(* PLC project mtcs_telemetry, Institute of Astronomy Onto 0.0.1 *)
(* stored: creationDateTime 2024-10-01T22:53:32.010142, modificationDateTime 2024-10-01T22:53:32.010142 *)

TYPE TelemetryParts : STRUCT
  temperatures : TelemetryTemperatures;  (* All temperature measurements *)
  relativeHumidities : TelemetryRelativeHumidities;  (* All relative humidity measurements *)
  dewpoints : TelemetryDewpoints;  (* All calculated dewpoints *)
  accelerometers : TelemetryAccelerometers;  (* Feedback from the accelerometers (vibrations + angles) *)
  io : TelemetryIO;  (* I/O modules *)
  flatfieldLeds : TelemetryFlatfieldLeds;  (* I/O modules *)
  configManager : ConfigManager;  (* The config manager (to load/save/activate configuration data) *)
END_STRUCT;
END_TYPE

TYPE TelemetryFlatfieldLedsParts : STRUCT
  output1 : SimpleRelay;  (* Output 1 *)
  output2 : SimpleRelay;  (* Output 2 *)
  output3 : SimpleRelay;  (* Output 3 *)
  output4 : SimpleRelay;  (* Output 4 *)
  output5 : SimpleRelay;  (* Output 5 *)
  output6 : SimpleRelay;  (* Output 6 *)
  output7 : SimpleRelay;  (* Output 7 *)
  output8 : SimpleRelay;  (* Output 8 *)
END_STRUCT;
END_TYPE

TYPE TelemetryIOParts : STRUCT
  coupler : EtherCatDevice;  (* Coupler *)
  slot5 : EtherCatDevice;  (* Slot 5 *)
  slot6 : EtherCatDevice;  (* Slot 6 *)
  slot7 : EtherCatDevice;  (* Slot 7 *)
  slot8 : EtherCatDevice;  (* Slot 8 *)
  slot9 : EtherCatDevice;  (* Slot 9 *)
  slot10 : EtherCatDevice;  (* Slot 10 *)
  slot11 : EtherCatDevice;  (* Slot 11 *)
  slot12 : EtherCatDevice;  (* Slot 12 *)
  slot13 : EtherCatDevice;  (* Slot 13 *)
  tubeAccelerometers : EtherCatDevice;  (* Tube accelerometers *)
END_STRUCT;
END_TYPE

TYPE TelemetryProcesses : STRUCT
  initialize : Process;  (* Start initializing *)
  lock : Process;  (* Lock the system *)
  unlock : Process;  (* Unlock the system *)
  changeOperatingState : ChangeOperatingStateProcess;  (* Change the operating state (e.g. AUTO, MANUAL, ...) *)
END_STRUCT;
END_TYPE

TYPE TelemetryTemperaturesStatuses : STRUCT
  healthStatus : HealthStatus;  (* Are all temperatures in a healthy state? *)
END_STRUCT;
END_TYPE

TYPE TelemetryRelativeHumiditiesStatuses : STRUCT
  healthStatus : HealthStatus;  (* Are all relative humidities in a healthy state? *)
END_STRUCT;
END_TYPE

TYPE TelemetryDewpointStatuses : STRUCT
  enabledStatus : EnabledStatus;  (* Is the dewpoint being calculated? *)
  healthStatus : HealthStatus;  (* Is the depoint OK? *)
  alarmStatus : HiHiLoLoAlarmStatus;  (* Alarm status *)
END_STRUCT;
END_TYPE

TYPE TelemetryDewpointsStatuses : STRUCT
  healthStatus : HealthStatus;  (* Are all dewpoints in a healthy state? *)
END_STRUCT;
END_TYPE

TYPE TelemetryAccelerometerStatuses : STRUCT
  xEnabledStatus : EnabledStatus;  (* Is the X angle being measured? *)
  yEnabledStatus : EnabledStatus;  (* Is the Y angle being measured? *)
  xHealthStatus : HealthStatus;  (* Is the X angle measurement OK? *)
  yHealthStatus : HealthStatus;  (* Is the Y angle measurement OK? *)
  xAlarmStatus : HiHiLoLoAlarmStatus;  (* Alarm status of the X angle *)
  yAlarmStatus : HiHiLoLoAlarmStatus;  (* Alarm status of the Y angle *)
END_STRUCT;
END_TYPE

TYPE TelemetryAccelerometersStatuses : STRUCT
  healthStatus : HealthStatus;  (* Are all accelerometers in a healthy state? *)
END_STRUCT;
END_TYPE

TYPE TelemetryStatuses : STRUCT
  initializationStatus : InitializationStatus;
  healthStatus : HealthStatus;
  busyStatus : BusyStatus;
  operatingStatus : OperatingStatus;
END_STRUCT;
END_TYPE

TYPE TelemetryFlatfieldLedsStatuses : STRUCT
  busyStatus : BusyStatus;
END_STRUCT;
END_TYPE

TYPE TelemetryIOStatuses : STRUCT
  healthStatus : HealthStatus;  (* Is the I/O in a healthy state? *)
END_STRUCT;
END_TYPE

TYPE TelemetryTemperaturesConfig : STRUCT
  m1 : MeasurementConfig;  (* Temperature of M1 *)
  mirrorCell : MeasurementConfig;  (* Temperature of the mirror cell *)
  m2 : MeasurementConfig;  (* Temperature of M2 *)
  m2Electronics : MeasurementConfig;  (* Temperature of the M2 electricity *)
  topTube : MeasurementConfig;  (* Temperature of the top of the tube *)
  centreTube : MeasurementConfig;  (* Temperature of the centre of the tube *)
  fork : MeasurementConfig;  (* Temperature of the fork *)
  nasmythAir : MeasurementConfig;  (* Temperature of the air inside the Nasmyth focal station *)
  rem : MeasurementConfig;  (* Temperature inside the REM cabinet *)
  rpm : MeasurementConfig;  (* Temperature inside the RPM cabinet *)
  hermesTelescopeAdapter : MeasurementConfig;  (* Temperature inside the HERMES telescope adapter *)
  topAir : MeasurementConfig;  (* Temperature of the air at the top of the tube *)
  insideTube : MeasurementConfig;  (* Temperature of the air inside the tube *)
END_STRUCT;
END_TYPE

TYPE TelemetryRelativeHumiditiesConfig : STRUCT
  topAir : MeasurementConfig;  (* Relative humidity of the air at the top of the tube *)
  insideTube : MeasurementConfig;  (* Relative humidity of the air inside the tube *)
END_STRUCT;
END_TYPE

TYPE TelemetryDewpointsConfig : STRUCT
  topAir : MeasurementConfig;  (* Dewpoint of the air at the top of the tube *)
  insideTube : MeasurementConfig;  (* Dewpoint of the air inside the tube *)
END_STRUCT;
END_TYPE

TYPE TelemetryAccelerometerConfig : STRUCT
  x : MeasurementConfig;  (* X angle *)
  y : MeasurementConfig;  (* X angle *)
END_STRUCT;
END_TYPE

TYPE TelemetryAccelerometersConfig : STRUCT
  tube : TelemetryAccelerometerConfig;  (* Accelerometer box at the tube *)
END_STRUCT;
END_TYPE

TYPE TelemetryConfig : STRUCT
  temperatures : TelemetryTemperaturesConfig;  (* All temperatures *)
  relativeHumidities : TelemetryRelativeHumiditiesConfig;  (* All relative humidities *)
  dewpoints : TelemetryDewpointsConfig;  (* All dewpoints *)
  accelerometers : TelemetryAccelerometersConfig;  (* All accelerometers *)
END_STRUCT;
END_TYPE

FUNCTION_BLOCK SM_TelemetryTemperatures
  VAR_OUTPUT
    {attribute 'OPC.UA.DA' := '1'}
    {attribute 'OPC.UA.DA.Access' := '1'}
    actualStatus : STRING;  (* Current status description *)
    previousStatus : STRING;  (* Previous status description *)
    {attribute 'OPC.UA.DA' := '1'}
    {attribute 'OPC.UA.DA.Access' := '1'}
    m1 : TemperatureMeasurement;  (* Temperature of M1 *)
    {attribute 'OPC.UA.DA' := '1'}
    {attribute 'OPC.UA.DA.Access' := '1'}
    mirrorCell : TemperatureMeasurement;  (* Temperature of the mirror cell *)
    {attribute 'OPC.UA.DA' := '1'}
    {attribute 'OPC.UA.DA.Access' := '1'}
    m2 : TemperatureMeasurement;  (* Temperature of M2 *)
    {attribute 'OPC.UA.DA' := '1'}
    {attribute 'OPC.UA.DA.Access' := '1'}
    m2Electronics : TemperatureMeasurement;  (* Temperature of the M2 electricity *)
    {attribute 'OPC.UA.DA' := '1'}
    {attribute 'OPC.UA.DA.Access' := '1'}
    topTube : TemperatureMeasurement;  (* Temperature of the top of the tube *)
    {attribute 'OPC.UA.DA' := '1'}
    {attribute 'OPC.UA.DA.Access' := '1'}
    centreTube : TemperatureMeasurement;  (* Temperature of the centre of the tube *)
    {attribute 'OPC.UA.DA' := '1'}
    {attribute 'OPC.UA.DA.Access' := '1'}
    fork : TemperatureMeasurement;  (* Temperature of the fork *)
    {attribute 'OPC.UA.DA' := '1'}
    {attribute 'OPC.UA.DA.Access' := '1'}
    nasmythAir : TemperatureMeasurement;  (* Temperature of the air inside the Nasmyth focal station *)
    {attribute 'OPC.UA.DA' := '1'}
    {attribute 'OPC.UA.DA.Access' := '1'}
    rem : TemperatureMeasurement;  (* Temperature inside the REM cabinet *)
    {attribute 'OPC.UA.DA' := '1'}
    {attribute 'OPC.UA.DA.Access' := '1'}
    rpm : TemperatureMeasurement;  (* Temperature inside the RPM cabinet *)
    {attribute 'OPC.UA.DA' := '1'}
    {attribute 'OPC.UA.DA.Access' := '1'}
    hermesTelescopeAdapter : TemperatureMeasurement;  (* Temperature inside the HERMES telescope adapter *)
    {attribute 'OPC.UA.DA' := '1'}
    {attribute 'OPC.UA.DA.Access' := '1'}
    topAir : TemperatureMeasurement;  (* Temperature of the air at the top of the tube *)
    {attribute 'OPC.UA.DA' := '1'}
    {attribute 'OPC.UA.DA.Access' := '1'}
    insideTube : TemperatureMeasurement;  (* Temperature of the air inside the tube *)
    statuses : TelemetryTemperaturesStatuses;  (* Statuses of the state machine *)
  END_VAR
  VAR_IN_OUT
    {attribute 'OPC.UA.DA' := '0'}
    config : TelemetryTemperaturesConfig;  (* Configuration of the temperatures *)
  END_VAR

            m1( config := config.m1 );
mirrorCell( config := config.mirrorCell );
m2( config := config.m2 );
m2Electronics( config := config.m2Electronics );
topTube( config := config.topTube );
centreTube( config := config.centreTube );
fork( config := config.fork );
nasmythAir( config := config.nasmythAir );
rem( config := config.rem );
rpm( config := config.rpm );
hermesTelescopeAdapter( config := config.hermesTelescopeAdapter );
topAir( config := config.topAir );
insideTube( config := config.insideTube );
statuses.healthStatus(
    isGood := (m1.statuses.healthStatus.isGood OR m1.statuses.enabledStatus.disabled) AND ((mirrorCell.statuses.healthStatus.isGood OR mirrorCell.statuses.enabledStatus.disabled) AND ((m2.statuses.healthStatus.isGood OR m2.statuses.enabledStatus.disabled) AND ((m2Electronics.statuses.healthStatus.isGood OR m2Electronics.statuses.enabledStatus.disabled) AND ((topTube.statuses.healthStatus.isGood OR topTube.statuses.enabledStatus.disabled) AND ((centreTube.statuses.healthStatus.isGood OR centreTube.statuses.enabledStatus.disabled) AND ((fork.statuses.healthStatus.isGood OR fork.statuses.enabledStatus.disabled) AND ((nasmythAir.statuses.healthStatus.isGood OR nasmythAir.statuses.enabledStatus.disabled) AND ((rem.statuses.healthStatus.isGood OR rem.statuses.enabledStatus.disabled) AND ((rpm.statuses.healthStatus.isGood OR rpm.statuses.enabledStatus.disabled) AND ((hermesTelescopeAdapter.statuses.healthStatus.isGood OR hermesTelescopeAdapter.statuses.enabledStatus.disabled) AND ((topAir.statuses.healthStatus.isGood OR topAir.statuses.enabledStatus.disabled) AND (insideTube.statuses.healthStatus.isGood OR insideTube.statuses.enabledStatus.disabled)))))))))))),
    hasWarning := m1.statuses.healthStatus.hasWarning OR (mirrorCell.statuses.healthStatus.hasWarning OR (m2.statuses.healthStatus.hasWarning OR (m2Electronics.statuses.healthStatus.hasWarning OR (topTube.statuses.healthStatus.hasWarning OR (centreTube.statuses.healthStatus.hasWarning OR (fork.statuses.healthStatus.hasWarning OR (nasmythAir.statuses.healthStatus.hasWarning OR (rem.statuses.healthStatus.hasWarning OR (rpm.statuses.healthStatus.hasWarning OR (hermesTelescopeAdapter.statuses.healthStatus.hasWarning OR (topAir.statuses.healthStatus.hasWarning OR insideTube.statuses.healthStatus.hasWarning))))))))))));

          

{attribute 'TcRpcEnable' := '1'}
METHOD _log : BOOL
  VAR_INPUT
    name : STRING;  (* Name of this function block instance *)
  END_VAR
  VAR_IN_OUT
    buffer : LogBuffer;  (* Buffer to write all logging to *)
  END_VAR
  VAR
    subBuffer : LogBuffer;  (* Temporary buffer to write logging by parts (sub-statemachines) to *)
  END_VAR
                  LOGGER(
    name := name,
    actualStatus := THIS^.actualStatus,
    previousStatus := THIS^.previousStatus,
    buffer := buffer,
    subBuffer := subBuffer,
    pHealthStatus := ADR(THIS^.statuses.healthStatus));

                
END_METHOD
END_FUNCTION_BLOCK

FUNCTION_BLOCK SM_TelemetryRelativeHumidities
  VAR_OUTPUT
    {attribute 'OPC.UA.DA' := '1'}
    {attribute 'OPC.UA.DA.Access' := '1'}
    actualStatus : STRING;  (* Current status description *)
    previousStatus : STRING;  (* Previous status description *)
    {attribute 'OPC.UA.DA' := '1'}
    {attribute 'OPC.UA.DA.Access' := '1'}
    topAir : RelativeHumidityMeasurement;  (* Relative humidity of the air at the top of the tube *)
    {attribute 'OPC.UA.DA' := '1'}
    {attribute 'OPC.UA.DA.Access' := '1'}
    insideTube : RelativeHumidityMeasurement;  (* Relative humidity of the air inside the tube *)
    statuses : TelemetryRelativeHumiditiesStatuses;  (* Statuses of the state machine *)
  END_VAR
  VAR_IN_OUT
    {attribute 'OPC.UA.DA' := '0'}
    config : TelemetryRelativeHumiditiesConfig;  (* Configuration of the relative humidities *)
  END_VAR

            topAir( config := config.topAir );
insideTube( config := config.insideTube );
statuses.healthStatus(
    isGood := (topAir.statuses.healthStatus.isGood OR topAir.statuses.enabledStatus.disabled) AND (insideTube.statuses.healthStatus.isGood OR insideTube.statuses.enabledStatus.disabled),
    hasWarning := topAir.statuses.healthStatus.hasWarning OR insideTube.statuses.healthStatus.hasWarning);

          

{attribute 'TcRpcEnable' := '1'}
METHOD _log : BOOL
  VAR_INPUT
    name : STRING;  (* Name of this function block instance *)
  END_VAR
  VAR_IN_OUT
    buffer : LogBuffer;  (* Buffer to write all logging to *)
  END_VAR
  VAR
    subBuffer : LogBuffer;  (* Temporary buffer to write logging by parts (sub-statemachines) to *)
  END_VAR
                  LOGGER(
    name := name,
    actualStatus := THIS^.actualStatus,
    previousStatus := THIS^.previousStatus,
    buffer := buffer,
    subBuffer := subBuffer,
    pHealthStatus := ADR(THIS^.statuses.healthStatus));

                
END_METHOD
END_FUNCTION_BLOCK

FUNCTION_BLOCK SM_TelemetryDewpoint
  VAR_OUTPUT
    {attribute 'OPC.UA.DA' := '1'}
    {attribute 'OPC.UA.DA.Access' := '1'}
    actualStatus : STRING;  (* Current status description *)
    previousStatus : STRING;  (* Previous status description *)
    {attribute 'OPC.UA.DA' := '1'}
    {attribute 'OPC.UA.DA.Access' := '1'}
    actual : Temperature;  (* Actual dewpoint temperature *)
    {attribute 'OPC.UA.DA' := '1'}
    {attribute 'OPC.UA.DA.Access' := '1'}
    average : Temperature;  (* Average dewpoint temperature *)
    statuses : TelemetryDewpointStatuses;  (* Statuses of the state machine *)
  END_VAR
  VAR_IN_OUT
    {attribute 'OPC.UA.DA' := '0'}
    config : MeasurementConfig;  (* Configuration *)
    {attribute 'OPC.UA.DA' := '0'}
    temperature : TemperatureMeasurement;  (* Temperature to be taken into account *)
    {attribute 'OPC.UA.DA' := '0'}
    relativeHumidity : RelativeHumidityMeasurement;  (* Relative humidity to be taken into account *)
  END_VAR

            statuses.enabledStatus( isEnabled := config.enabled );
statuses.healthStatus(
    superState := statuses.enabledStatus.enabled,
    isGood := NOT(temperature.error OR (relativeHumidity.statuses.healthStatus.bad OR (statuses.alarmStatus.hiHi OR statuses.alarmStatus.loLo))),
    hasWarning := statuses.alarmStatus.hi OR statuses.alarmStatus.lo);
statuses.alarmStatus(
    superState := statuses.enabledStatus.enabled,
    config := config.alarms,
    value := average.celsius.value);

          

{attribute 'TcRpcEnable' := '1'}
METHOD _log : BOOL
  VAR_INPUT
    name : STRING;  (* Name of this function block instance *)
  END_VAR
  VAR_IN_OUT
    buffer : LogBuffer;  (* Buffer to write all logging to *)
  END_VAR
  VAR
    subBuffer : LogBuffer;  (* Temporary buffer to write logging by parts (sub-statemachines) to *)
  END_VAR
                  LOGGER(
    name := name,
    actualStatus := THIS^.actualStatus,
    previousStatus := THIS^.previousStatus,
    buffer := buffer,
    subBuffer := subBuffer,
    pHealthStatus := ADR(THIS^.statuses.healthStatus));

                
END_METHOD
END_FUNCTION_BLOCK

FUNCTION_BLOCK SM_TelemetryDewpoints
  VAR_OUTPUT
    {attribute 'OPC.UA.DA' := '1'}
    {attribute 'OPC.UA.DA.Access' := '1'}
    actualStatus : STRING;  (* Current status description *)
    previousStatus : STRING;  (* Previous status description *)
    {attribute 'OPC.UA.DA' := '1'}
    {attribute 'OPC.UA.DA.Access' := '1'}
    topAir : TelemetryDewpoint;  (* Dewpoint of the air at the top of the tube *)
    {attribute 'OPC.UA.DA' := '1'}
    {attribute 'OPC.UA.DA.Access' := '1'}
    insideTube : TelemetryDewpoint;  (* Dewpoint of the air inside the tube *)
    statuses : TelemetryDewpointsStatuses;  (* Statuses of the state machine *)
  END_VAR
  VAR_IN_OUT
    {attribute 'OPC.UA.DA' := '0'}
    config : TelemetryDewpointsConfig;  (* Configuration of the dewpoints *)
    {attribute 'OPC.UA.DA' := '0'}
    temperatures : TelemetryTemperatures;  (* Measured temperatures *)
    {attribute 'OPC.UA.DA' := '0'}
    relativeHumidities : TelemetryRelativeHumidities;  (* Measured relative humidities *)
  END_VAR

            topAir(
    config := config.topAir,
    temperature := temperatures.topAir,
    relativeHumidity := relativeHumidities.topAir);
insideTube(
    config := config.insideTube,
    temperature := temperatures.insideTube,
    relativeHumidity := relativeHumidities.insideTube);
statuses.healthStatus(
    isGood := (topAir.statuses.healthStatus.isGood OR topAir.statuses.enabledStatus.disabled) AND (insideTube.statuses.healthStatus.isGood OR insideTube.statuses.enabledStatus.disabled),
    hasWarning := topAir.statuses.healthStatus.hasWarning OR insideTube.statuses.healthStatus.hasWarning);

          

{attribute 'TcRpcEnable' := '1'}
METHOD _log : BOOL
  VAR_INPUT
    name : STRING;  (* Name of this function block instance *)
  END_VAR
  VAR_IN_OUT
    buffer : LogBuffer;  (* Buffer to write all logging to *)
  END_VAR
  VAR
    subBuffer : LogBuffer;  (* Temporary buffer to write logging by parts (sub-statemachines) to *)
  END_VAR
                  LOGGER(
    name := name,
    actualStatus := THIS^.actualStatus,
    previousStatus := THIS^.previousStatus,
    buffer := buffer,
    subBuffer := subBuffer,
    pHealthStatus := ADR(THIS^.statuses.healthStatus));

                
END_METHOD
END_FUNCTION_BLOCK

FUNCTION_BLOCK SM_TelemetryAccelerometer
  VAR_OUTPUT
    {attribute 'OPC.UA.DA' := '1'}
    {attribute 'OPC.UA.DA.Access' := '1'}
    actualStatus : STRING;  (* Current status description *)
    previousStatus : STRING;  (* Previous status description *)
    {attribute 'OPC.UA.DA' := '1'}
    {attribute 'OPC.UA.DA.Access' := '1'}
    X1plus : GForceMeasurement;  (* +X1 (channel 1 of EP1816-3008) *)
    {attribute 'OPC.UA.DA' := '1'}
    {attribute 'OPC.UA.DA.Access' := '1'}
    Y1plus : GForceMeasurement;  (* +Y1 (channel 2 of EP1816-3008) *)
    {attribute 'OPC.UA.DA' := '1'}
    {attribute 'OPC.UA.DA.Access' := '1'}
    Z1minus : GForceMeasurement;  (* -Z1 (channel 3 of EP1816-3008) *)
    {attribute 'OPC.UA.DA' := '1'}
    {attribute 'OPC.UA.DA.Access' := '1'}
    Y2plus : GForceMeasurement;  (* +Y2 (channel 4 of EP1816-3008) *)
    {attribute 'OPC.UA.DA' := '1'}
    {attribute 'OPC.UA.DA.Access' := '1'}
    X2minus : GForceMeasurement;  (* -X2 (channel 5 of EP1816-3008) *)
    {attribute 'OPC.UA.DA' := '1'}
    {attribute 'OPC.UA.DA.Access' := '1'}
    Z2minus : GForceMeasurement;  (* -Z2 (channel 6 of EP1816-3008) *)
    {attribute 'OPC.UA.DA' := '1'}
    {attribute 'OPC.UA.DA.Access' := '1'}
    actualXAngle : AngularPosition;  (* Actual X angle *)
    {attribute 'OPC.UA.DA' := '1'}
    {attribute 'OPC.UA.DA.Access' := '1'}
    actualYAngle : AngularPosition;  (* Actual Y angle *)
    {attribute 'OPC.UA.DA' := '1'}
    {attribute 'OPC.UA.DA.Access' := '1'}
    averageXAngle : AngularPosition;  (* Average X angle *)
    {attribute 'OPC.UA.DA' := '1'}
    {attribute 'OPC.UA.DA.Access' := '1'}
    averageYAngle : AngularPosition;  (* Average Y angle *)
    statuses : TelemetryAccelerometerStatuses;  (* Statuses of the state machine *)
  END_VAR
  VAR_IN_OUT
    {attribute 'OPC.UA.DA' := '0'}
    xConfig : MeasurementConfig;  (* Reference to the config of the X angle (alarms in degrees) *)
    {attribute 'OPC.UA.DA' := '0'}
    yConfig : MeasurementConfig;  (* Reference to the config of the Y angle (alarms in degrees) *)
  END_VAR

            statuses.xEnabledStatus( isEnabled := xConfig.enabled );
statuses.yEnabledStatus( isEnabled := yConfig.enabled );
statuses.xHealthStatus(
    superState := statuses.xEnabledStatus.enabled,
    isGood := NOT(statuses.xAlarmStatus.hiHi OR statuses.xAlarmStatus.loLo),
    hasWarning := statuses.xAlarmStatus.hi OR statuses.xAlarmStatus.lo);
statuses.yHealthStatus(
    superState := statuses.yEnabledStatus.enabled,
    isGood := NOT(statuses.yAlarmStatus.hiHi OR statuses.yAlarmStatus.loLo),
    hasWarning := statuses.yAlarmStatus.hi OR statuses.yAlarmStatus.lo);
statuses.xAlarmStatus(
    superState := statuses.xEnabledStatus.enabled,
    config := xConfig.alarms,
    value := averageXAngle.degrees.value);
statuses.yAlarmStatus(
    superState := statuses.yEnabledStatus.enabled,
    config := yConfig.alarms,
    value := averageYAngle.degrees.value);

          

{attribute 'TcRpcEnable' := '1'}
METHOD _log : BOOL
  VAR_INPUT
    name : STRING;  (* Name of this function block instance *)
  END_VAR
  VAR_IN_OUT
    buffer : LogBuffer;  (* Buffer to write all logging to *)
  END_VAR
  VAR
    subBuffer : LogBuffer;  (* Temporary buffer to write logging by parts (sub-statemachines) to *)
  END_VAR
                  LOGGER(
    name := name,
    actualStatus := THIS^.actualStatus,
    previousStatus := THIS^.previousStatus,
    buffer := buffer,
    subBuffer := subBuffer);

                
END_METHOD
END_FUNCTION_BLOCK

FUNCTION_BLOCK SM_TelemetryAccelerometers
  VAR_OUTPUT
    {attribute 'OPC.UA.DA' := '1'}
    {attribute 'OPC.UA.DA.Access' := '1'}
    actualStatus : STRING;  (* Current status description *)
    previousStatus : STRING;  (* Previous status description *)
    {attribute 'OPC.UA.DA' := '1'}
    {attribute 'OPC.UA.DA.Access' := '1'}
    tube : TelemetryAccelerometer;  (* Accelerometer box at the tube *)
    statuses : TelemetryAccelerometersStatuses;  (* Statuses of the state machine *)
  END_VAR
  VAR_IN_OUT
    {attribute 'OPC.UA.DA' := '0'}
    config : TelemetryAccelerometersConfig;  (* Configuration of the accelerometers *)
  END_VAR

            tube(
    xConfig := config.tube.x,
    yConfig := config.tube.y);
statuses.healthStatus(
    isGood := tube.statuses.xHealthStatus.isGood AND tube.statuses.yHealthStatus.isGood,
    hasWarning := tube.statuses.xHealthStatus.hasWarning OR tube.statuses.yHealthStatus.hasWarning);

          

{attribute 'TcRpcEnable' := '1'}
METHOD _log : BOOL
  VAR_INPUT
    name : STRING;  (* Name of this function block instance *)
  END_VAR
  VAR_IN_OUT
    buffer : LogBuffer;  (* Buffer to write all logging to *)
  END_VAR
  VAR
    subBuffer : LogBuffer;  (* Temporary buffer to write logging by parts (sub-statemachines) to *)
  END_VAR
                  LOGGER(
    name := name,
    actualStatus := THIS^.actualStatus,
    previousStatus := THIS^.previousStatus,
    buffer := buffer,
    subBuffer := subBuffer,
    pHealthStatus := ADR(THIS^.statuses.healthStatus));

                
END_METHOD
END_FUNCTION_BLOCK

FUNCTION_BLOCK SM_Telemetry
  VAR_INPUT
    {attribute 'OPC.UA.DA' := '1'}
    {attribute 'OPC.UA.DA.Access' := '1'}
    editableConfig : TelemetryConfig;  (* Editable configuration of the Telemetry subsystem *)
  END_VAR
  VAR_OUTPUT
    {attribute 'OPC.UA.DA' := '1'}
    {attribute 'OPC.UA.DA.Access' := '1'}
    actualStatus : STRING;  (* Current status description *)
    previousStatus : STRING;  (* Previous status description *)
    {attribute 'OPC.UA.DA' := '1'}
    {attribute 'OPC.UA.DA.Access' := '1'}
    config : TelemetryConfig;  (* Active configuration of the Telemetry subsystem *)
    statuses : TelemetryStatuses;  (* Statuses of the state machine *)
    parts : TelemetryParts;  (* Parts of the state machine *)
    processes : TelemetryProcesses;  (* Processes of the state machine *)
  END_VAR
  VAR_IN_OUT
    {attribute 'OPC.UA.DA' := '0'}
    operatorStatus : OperatorStatus;  (* Shared operator status *)
  END_VAR

            parts.temperatures( config := config.temperatures );
parts.relativeHumidities( config := config.relativeHumidities );
parts.dewpoints(
    config := config.dewpoints,
    temperatures := parts.temperatures,
    relativeHumidities := parts.relativeHumidities);
parts.accelerometers( config := config.accelerometers );
parts.io();
parts.flatfieldLeds( isEnabled := statuses.initializationStatus.initialized AND statuses.operatingStatus.manual );
parts.configManager( isEnabled := operatorStatus.tech );
statuses.initializationStatus();
statuses.healthStatus(
    isGood := parts.temperatures.statuses.healthStatus.isGood AND (parts.relativeHumidities.statuses.healthStatus.isGood AND (parts.dewpoints.statuses.healthStatus.isGood AND (parts.accelerometers.statuses.healthStatus.isGood AND (parts.io.statuses.healthStatus.isGood AND parts.configManager.statuses.healthStatus.isGood)))),
    hasWarning := parts.temperatures.statuses.healthStatus.hasWarning OR (parts.relativeHumidities.statuses.healthStatus.hasWarning OR (parts.dewpoints.statuses.healthStatus.hasWarning OR (parts.accelerometers.statuses.healthStatus.hasWarning OR (parts.io.statuses.healthStatus.hasWarning OR parts.configManager.statuses.healthStatus.hasWarning)))));
statuses.busyStatus( isBusy := statuses.initializationStatus.initializing OR (parts.flatfieldLeds.statuses.busyStatus.busy OR parts.configManager.statuses.busyStatus.busy) );
statuses.operatingStatus( superState := statuses.initializationStatus.initialized );
processes.initialize( isEnabled := statuses.initializationStatus.shutdown OR (statuses.initializationStatus.initializingFailed OR statuses.initializationStatus.initialized) );
processes.lock( isEnabled := operatorStatus.tech AND statuses.initializationStatus.initialized );
processes.unlock( isEnabled := operatorStatus.tech AND statuses.initializationStatus.locked );
processes.changeOperatingState( isEnabled := statuses.busyStatus.idle AND statuses.initializationStatus.initialized );

          

{attribute 'TcRpcEnable' := '1'}
METHOD initialize : RequestResults
                  initialize := THIS^.processes.initialize.request();

                
END_METHOD

{attribute 'TcRpcEnable' := '1'}
METHOD lock : RequestResults
                  lock := THIS^.processes.lock.request();

                
END_METHOD

{attribute 'TcRpcEnable' := '1'}
METHOD unlock : RequestResults
                  unlock := THIS^.processes.unlock.request();

                
END_METHOD

{attribute 'TcRpcEnable' := '1'}
METHOD changeOperatingState : RequestResults
  VAR_INPUT
    state : OperatingStates;
  END_VAR
                  changeOperatingState := THIS^.processes.changeOperatingState.request( state := state );

                
END_METHOD

{attribute 'TcRpcEnable' := '1'}
METHOD _log : BOOL
  VAR_INPUT
    name : STRING;  (* Name of this function block instance *)
  END_VAR
  VAR_IN_OUT
    buffer : LogBuffer;  (* Buffer to write all logging to *)
  END_VAR
  VAR
    subBuffer : LogBuffer;  (* Temporary buffer to write logging by parts (sub-statemachines) to *)
  END_VAR
                  THIS^.parts.temperatures._log(
    name := 'temperatures',
    buffer := subBuffer);
THIS^.parts.relativeHumidities._log(
    name := 'relativeHumidities',
    buffer := subBuffer);
THIS^.parts.dewpoints._log(
    name := 'dewpoints',
    buffer := subBuffer);
THIS^.parts.accelerometers._log(
    name := 'accelerometers',
    buffer := subBuffer);
THIS^.parts.io._log(
    name := 'io',
    buffer := subBuffer);
THIS^.parts.flatfieldLeds._log(
    name := 'flatfieldLeds',
    buffer := subBuffer);
THIS^.parts.configManager._log(
    name := 'configManager',
    buffer := subBuffer);
THIS^.processes.initialize._log(
    name := 'processes.initialize',
    buffer := subBuffer);
THIS^.processes.lock._log(
    name := 'processes.lock',
    buffer := subBuffer);
THIS^.processes.unlock._log(
    name := 'processes.unlock',
    buffer := subBuffer);
THIS^.processes.changeOperatingState._log(
    name := 'processes.changeOperatingState',
    buffer := subBuffer);
LOGGER(
    name := name,
    actualStatus := THIS^.actualStatus,
    previousStatus := THIS^.previousStatus,
    buffer := buffer,
    subBuffer := subBuffer,
    pHealthStatus := ADR(THIS^.statuses.healthStatus),
    pBusyStatus := ADR(THIS^.statuses.busyStatus));

                
END_METHOD
END_FUNCTION_BLOCK

FUNCTION_BLOCK SM_TelemetryFlatfieldLeds
  VAR_INPUT
    {attribute 'OPC.UA.DA' := '0'}
    isEnabled : BOOL;  (* Is control enabled? *)
  END_VAR
  VAR_OUTPUT
    {attribute 'OPC.UA.DA' := '1'}
    {attribute 'OPC.UA.DA.Access' := '1'}
    actualStatus : STRING;  (* Current status description *)
    previousStatus : STRING;  (* Previous status description *)
    statuses : TelemetryFlatfieldLedsStatuses;  (* Statuses of the state machine *)
    parts : TelemetryFlatfieldLedsParts;  (* Parts of the state machine *)
  END_VAR

            parts.output1( isEnabled := isEnabled );
parts.output2( isEnabled := isEnabled );
parts.output3( isEnabled := isEnabled );
parts.output4( isEnabled := isEnabled );
parts.output5( isEnabled := isEnabled );
parts.output6( isEnabled := isEnabled );
parts.output7( isEnabled := isEnabled );
parts.output8( isEnabled := isEnabled );
statuses.busyStatus( isBusy := parts.output1.statuses.busyStatus.busy OR (parts.output2.statuses.busyStatus.busy OR (parts.output3.statuses.busyStatus.busy OR (parts.output4.statuses.busyStatus.busy OR (parts.output5.statuses.busyStatus.busy OR (parts.output6.statuses.busyStatus.busy OR (parts.output7.statuses.busyStatus.busy OR parts.output8.statuses.busyStatus.busy)))))) );

          

{attribute 'TcRpcEnable' := '1'}
METHOD _log : BOOL
  VAR_INPUT
    name : STRING;  (* Name of this function block instance *)
  END_VAR
  VAR_IN_OUT
    buffer : LogBuffer;  (* Buffer to write all logging to *)
  END_VAR
  VAR
    subBuffer : LogBuffer;  (* Temporary buffer to write logging by parts (sub-statemachines) to *)
  END_VAR
                  THIS^.parts.output1._log(
    name := 'output1',
    buffer := subBuffer);
THIS^.parts.output2._log(
    name := 'output2',
    buffer := subBuffer);
THIS^.parts.output3._log(
    name := 'output3',
    buffer := subBuffer);
THIS^.parts.output4._log(
    name := 'output4',
    buffer := subBuffer);
THIS^.parts.output5._log(
    name := 'output5',
    buffer := subBuffer);
THIS^.parts.output6._log(
    name := 'output6',
    buffer := subBuffer);
THIS^.parts.output7._log(
    name := 'output7',
    buffer := subBuffer);
THIS^.parts.output8._log(
    name := 'output8',
    buffer := subBuffer);
LOGGER(
    name := name,
    actualStatus := THIS^.actualStatus,
    previousStatus := THIS^.previousStatus,
    buffer := buffer,
    subBuffer := subBuffer,
    pBusyStatus := ADR(THIS^.statuses.busyStatus));

                
END_METHOD
END_FUNCTION_BLOCK

FUNCTION_BLOCK SM_TelemetryIO
  VAR_OUTPUT
    {attribute 'OPC.UA.DA' := '1'}
    {attribute 'OPC.UA.DA.Access' := '1'}
    actualStatus : STRING;  (* Current status description *)
    previousStatus : STRING;  (* Previous status description *)
    statuses : TelemetryIOStatuses;  (* Statuses of the state machine *)
    parts : TelemetryIOParts;  (* Parts of the state machine *)
  END_VAR

            parts.coupler(
    id := 'COUPLER',
    typeId := 'EK1100');
parts.slot5(
    id := '113A1',
    typeId := 'EL3202-0010');
parts.slot6(
    id := '114A1',
    typeId := 'EL3202-0010');
parts.slot7(
    id := '115A1',
    typeId := 'EL3202-0010');
parts.slot8(
    id := '116A1',
    typeId := 'EL3202-0010');
parts.slot9(
    id := '117A1',
    typeId := 'EL3202-0010');
parts.slot10(
    id := '118A1',
    typeId := 'EL3202-0010');
parts.slot11(
    id := '119A1',
    typeId := 'EL3202-0010');
parts.slot12(
    id := '120A1',
    typeId := 'EL3024');
parts.slot13(
    id := '121A1',
    typeId := 'EL2008');
parts.tubeAccelerometers(
    id := 'ACCTUB',
    typeId := 'EP1816-3008');
statuses.healthStatus( isGood := parts.coupler.statuses.healthStatus.isGood AND (parts.slot5.statuses.healthStatus.isGood AND (parts.slot6.statuses.healthStatus.isGood AND (parts.slot7.statuses.healthStatus.isGood AND (parts.slot8.statuses.healthStatus.isGood AND (parts.slot9.statuses.healthStatus.isGood AND (parts.slot10.statuses.healthStatus.isGood AND (parts.slot11.statuses.healthStatus.isGood AND (parts.slot12.statuses.healthStatus.isGood AND (parts.slot13.statuses.healthStatus.isGood AND parts.tubeAccelerometers.statuses.healthStatus.isGood))))))))) );

          

{attribute 'TcRpcEnable' := '1'}
METHOD _log : BOOL
  VAR_INPUT
    name : STRING;  (* Name of this function block instance *)
  END_VAR
  VAR_IN_OUT
    buffer : LogBuffer;  (* Buffer to write all logging to *)
  END_VAR
  VAR
    subBuffer : LogBuffer;  (* Temporary buffer to write logging by parts (sub-statemachines) to *)
  END_VAR
                  THIS^.parts.coupler._log(
    name := 'coupler',
    buffer := subBuffer);
THIS^.parts.slot5._log(
    name := 'slot5',
    buffer := subBuffer);
THIS^.parts.slot6._log(
    name := 'slot6',
    buffer := subBuffer);
THIS^.parts.slot7._log(
    name := 'slot7',
    buffer := subBuffer);
THIS^.parts.slot8._log(
    name := 'slot8',
    buffer := subBuffer);
THIS^.parts.slot9._log(
    name := 'slot9',
    buffer := subBuffer);
THIS^.parts.slot10._log(
    name := 'slot10',
    buffer := subBuffer);
THIS^.parts.slot11._log(
    name := 'slot11',
    buffer := subBuffer);
THIS^.parts.slot12._log(
    name := 'slot12',
    buffer := subBuffer);
THIS^.parts.slot13._log(
    name := 'slot13',
    buffer := subBuffer);
THIS^.parts.tubeAccelerometers._log(
    name := 'tubeAccelerometers',
    buffer := subBuffer);
LOGGER(
    name := name,
    actualStatus := THIS^.actualStatus,
    previousStatus := THIS^.previousStatus,
    buffer := buffer,
    subBuffer := subBuffer,
    pHealthStatus := ADR(THIS^.statuses.healthStatus));

                
END_METHOD
END_FUNCTION_BLOCK
